// Mitsubishi GX Works2 project: 2023-05-09 #1   PLC: Q03UDV
// 생산자동화기능사

// global labels: Global1
VAR_GLOBAL
  PB1 AT X0 : BOOL;
  PB2 AT X1 : BOOL;
  정지 AT X2 : BOOL;
  공급후진 AT X3 : BOOL;
  공급전진 AT X4 : BOOL;
  가공후진 AT X5 : BOOL;
  가공전진 AT X6 : BOOL;
  송출후진 AT X7 : BOOL;
  송출전진 AT X8 : BOOL;
  배출후진 AT X9 : BOOL;
  배출전진 AT X0A : BOOL;
  매거진 AT X0B : BOOL;
  금속 AT X0F : BOOL;
  적색 AT Y20 : BOOL;
  황색 AT Y21 : BOOL;
  녹색 AT Y22 : BOOL;
  공급1 AT Y23 : BOOL;
  공급2 AT Y24 : BOOL;
  가공 AT Y25 : BOOL;
  드릴 AT Y26 : BOOL;
  송출 AT Y27 : BOOL;
  배출 AT Y28 : BOOL;
  컨베이어 AT Y29 : BOOL;
  PB3 AT X0C : BOOL;
END_VAR

PROGRAM 기본동작
VAR
  STATE : INT;
END_VAR
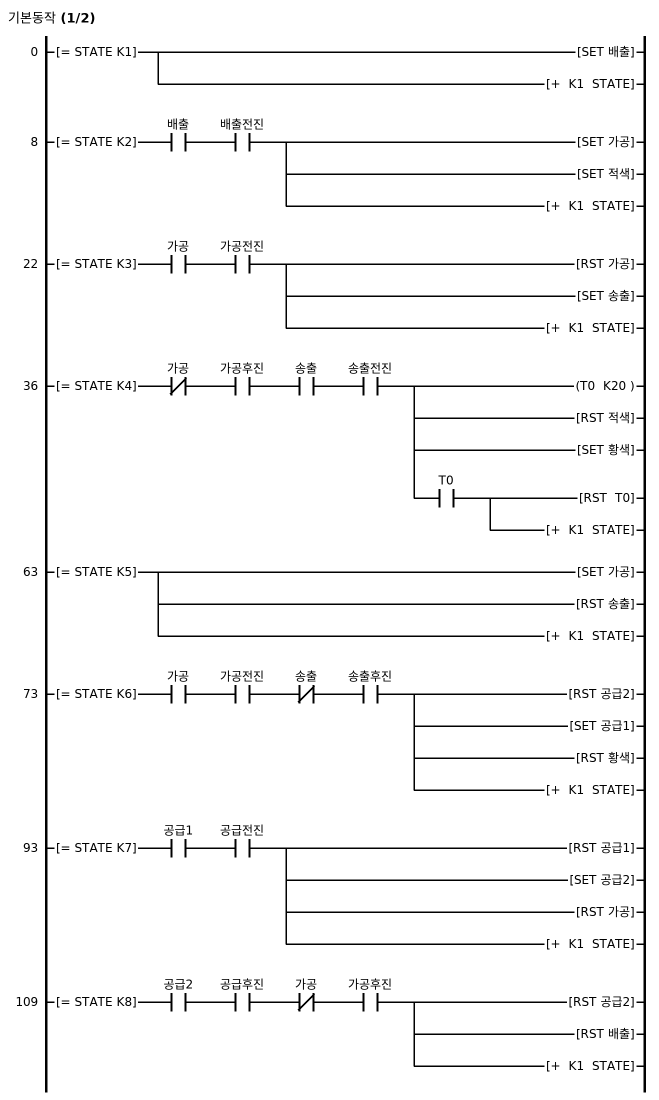
0     LD=     STATE K1
      SET     배출
      +       K1 STATE
8     LD=     STATE K2
      AND     배출
      AND     배출전진
      SET     가공
      SET     적색
      +       K1 STATE
22    LD=     STATE K3
      AND     가공
      AND     가공전진
      RST     가공
      SET     송출
      +       K1 STATE
36    LD=     STATE K4
      ANI     가공
      AND     가공후진
      AND     송출
      AND     송출전진
      OUT     T0 K20
      RST     적색
      SET     황색
      AND     T0
      RST     T0
      +       K1 STATE
63    LD=     STATE K5
      SET     가공
      RST     송출
      +       K1 STATE
73    LD=     STATE K6
      AND     가공
      AND     가공전진
      ANI     송출
      AND     송출후진
      RST     공급2
      SET     공급1
      RST     황색
      +       K1 STATE
93    LD=     STATE K7
      AND     공급1
      AND     공급전진
      RST     공급1
      SET     공급2
      RST     가공
      +       K1 STATE
109   LD=     STATE K8
      AND     공급2
      AND     공급후진
      ANI     가공
      AND     가공후진
      RST     공급2
      RST     배출
      +       K1 STATE
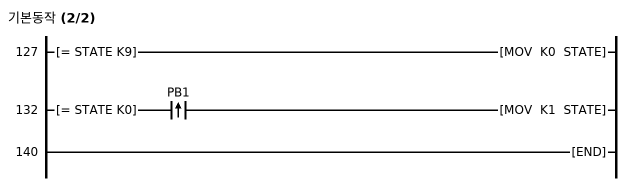
127   LD=     STATE K9
      MOV     K0 STATE
132   LD=     STATE K0
      ANDP    PB1
      MOV     K1 STATE
140   END
END_PROGRAM

PROGRAM 응용동작1
VAR
  STATE : INT;
  비금속 : BOOL;
END_VAR
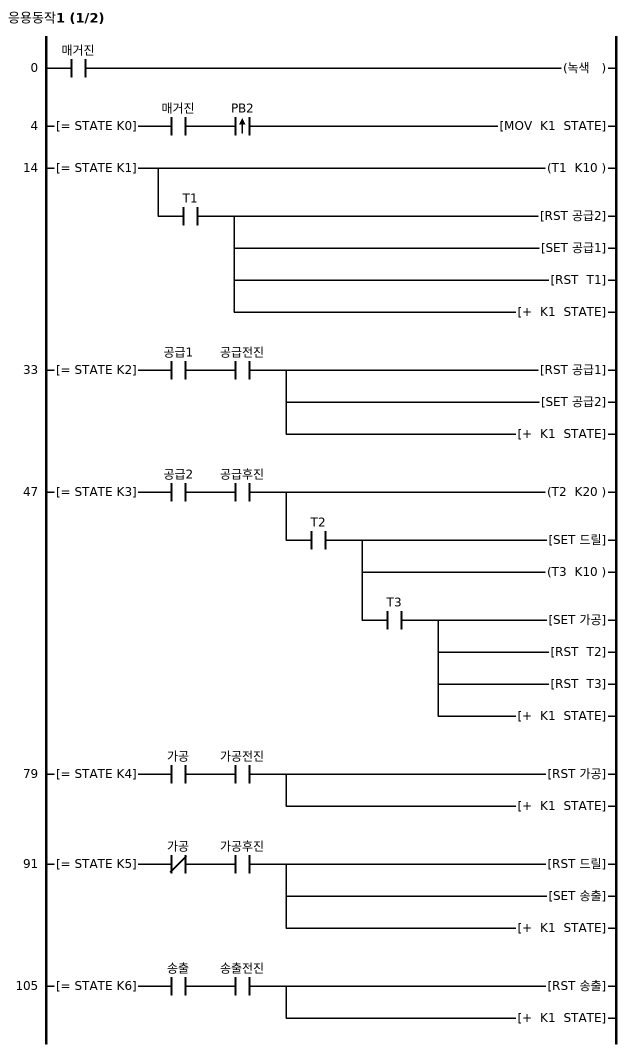
0     LD      매거진
      OUT     녹색
4     LD=     STATE K0
      AND     매거진
      ANDP    PB2
      MOV     K1 STATE
14    LD=     STATE K1
      OUT     T1 K10
      AND     T1
      RST     공급2
      SET     공급1
      RST     T1
      +       K1 STATE
33    LD=     STATE K2
      AND     공급1
      AND     공급전진
      RST     공급1
      SET     공급2
      +       K1 STATE
47    LD=     STATE K3
      AND     공급2
      AND     공급후진
      OUT     T2 K20
      AND     T2
      SET     드릴
      OUT     T3 K10
      AND     T3
      SET     가공
      RST     T2
      RST     T3
      +       K1 STATE
79    LD=     STATE K4
      AND     가공
      AND     가공전진
      RST     가공
      +       K1 STATE
91    LD=     STATE K5
      ANI     가공
      AND     가공후진
      RST     드릴
      SET     송출
      +       K1 STATE
105   LD=     STATE K6
      AND     송출
      AND     송출전진
      RST     송출
      +       K1 STATE
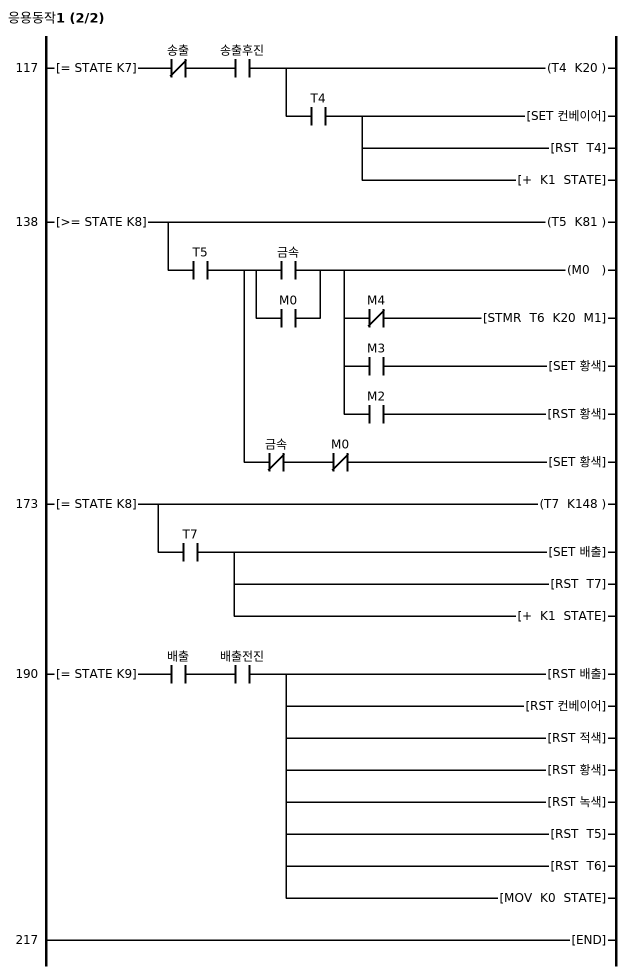
117   LD=     STATE K7
      ANI     송출
      AND     송출후진
      OUT     T4 K20
      AND     T4
      SET     컨베이어
      RST     T4
      +       K1 STATE
138   LD>=    STATE K8
      OUT     T5 K81
      AND     T5
      MPS
      LD      금속
      OR      M0
      ANB
      OUT     M0
      MPS
      ANI     M4
      STMR    T6 K20 M1
      MRD
      AND     M3
      SET     황색
      MPP
      AND     M2
      RST     황색
      MPP
      ANI     금속
      ANI     M0
      SET     황색
173   LD=     STATE K8
      OUT     T7 K148
      AND     T7
      SET     배출
      RST     T7
      +       K1 STATE
190   LD=     STATE K9
      AND     배출
      AND     배출전진
      RST     배출
      RST     컨베이어
      RST     적색
      RST     황색
      RST     녹색
      RST     T5
      RST     T6
      MOV     K0 STATE
217   END
END_PROGRAM
